Omron CX-Programmer project NewProject (CX-Programmer 9.87)

# PLC Teste: CP1L M

## Global symbols (name address type ; comment)
D315 CHANNEL  ; fim dm de contagem
Banco_de_Dados_29 Contador_de_Peças_PH29
Banco_de_Dados_30 Contador_de_Peças_PH30
Banco_de_Dados_31 Contador_de_Peças_PH31
Banco_de_Dados_F17 Contador_de_Peças_F17
Banco_de_Dados_F18 Contador_de_Peças_F18
Banco_de_Dados_F22 Contador_de_Peças_F22
Banco_de_Dados_R42 Contador_de_Peças_RC42
Banco_de_Dados_R43 Contador_de_Peças_RC43
Banco_de_dados_R41 Contador_de_Peças_RC41
Conta_Peças Contador_de_Peças_PH31
Visual_Formato_Trabalho_29 Formato_de_Trabalho_29
Visual_Formato_Trabalho_30 Formato_de_Trabalho_30
Visual_Formato_Trabalho_31 Formato_de_Trabalho_31

## Program Prensa (cyclic task 0)
Local symbols
F_31dias_vezes_2_ph30 D546 WORD
F_31dias_vezes_2_ph31 D530 WORD
F_Memoria_contagem_BCD_ph30 D552 WORD
F_Memoria_contagem_BCD_ph31 D536 WORD
F_Memória_de_Armazenagem_ph30 D550 WORD
F_Memória_de_Armazenagem_ph31 D534 WORD
F_Ponteiro_Dword_ph30 D548 WORD
F_Ponteiro_Dword_ph31 D532 WORD
KEEP 10.04 BOOL
MemAtuaReloSupervisorio H10.01 BOOL  ; Memória Atualiza Relogio pelo supervisório
Memoria_contagem_BCD_ph29 D528 WORD
Memoria_contagem_BCD_ph30 D518 WORD
Memoria_contagem_BCD_ph31 D508 WORD
Memoria_contagem_BIN_ph29 D526 WORD
Memoria_contagem_BIN_ph30 D516 WORD
Memoria_contagem_BIN_ph31 D506 WORD
Memória_de_Armazenagem_ph29 D524 WORD
Memória_de_Armazenagem_ph30 D514 WORD
Memória_de_Armazenagem_ph31 D504 WORD
PH29paradaT1 D0 CHANNEL  ; cnt prensa 31 parada T1
PH29paradaT2 D6 CHANNEL  ; cnt prensa 31 parada T2
PH29paradaT3 D12 CHANNEL  ; cnt prensa 31 parada T3
PH30paradaT1 D2 CHANNEL  ; cnt prensa 31 parada T1
PH30paradaT2 D8 CHANNEL  ; cnt prensa 31 parada T2
PH30paradaT3 D14 CHANNEL  ; cnt prensa 31 parada T3
PH31paradaT1 D4 CHANNEL  ; cnt prensa 31 parada T1
PH31paradaT2 D10 CHANNEL  ; cnt prensa 31 parada T2
PH31paradaT3 D18 CHANNEL  ; cnt prensa 31 parada T3
Ponteiro_Dword_ph29 D522 WORD
Ponteiro_Dword_ph30 D512 WORD
Ponteiro_Dword_ph31 D502 WORD
_31dias_vezes_2_ph29 D520 WORD
_31dias_vezes_2_ph30 D510 WORD
_31dias_vezes_2_ph31 D500 WORD
anoRelogio D36 CHANNEL  ; Ano Relógio
codFormPH29 D54 CHANNEL  ; Codigo do formato ph29
codFormPH30 D50 CHANNEL  ; Codigo do formato ph30
codFormPH31 D46 CHANNEL  ; Codigo do formato ph31
delayCicloPrensa29 T0001 BOOL  ; Retardo ciclo da prensa
delayCicloPrensa30 T0002 BOOL  ; Retardo ciclo da prensa
delayCicloPrensa31 T0003 BOOL  ; Retardo ciclo da prensa
diaCalendario D64 CHANNEL  ; dia calendario
diaMes D40 CHANNEL  ; dia do mes
diaRelogio D32 CHANNEL  ; Dia Relógio
filtroCntPc29 T0004 BOOL  ; filtro contagem peças
filtroCntPc30 T0005 BOOL  ; filtro contagem peças
filtroCntPc31 T0006 BOOL  ; filtro contagem peças
firstDMenvioFormat D56 CHANNEL  ; primeiro DM envio formato
firstDMenvioPcPH D42 CHANNEL  ; pirmeiro DM de envio peças ph
horaRelogio D30 CHANNEL  ; Horas Relogio
horas D58 CHANNEL  ; horas
iniciaCntTurno1 H10.02 BOOL  ; inicia contagem turno 1
iniciaCntTurno2 H10.03 BOOL  ; inicia contagem turno 2
iniciaCntTurno3 H10.04 BOOL  ; iniio contagem turno 3
linhaSelect D70 CHANNEL  ; linha selecionada
mesCalendario D66 CHANNEL  ; mes calendario
mesRelogio D34 CHANNEL  ; Mes Relogio
mesSelecionado D68 CHANNEL  ; mês selecionado
mesSelect D72 CHANNEL  ; mês selecionado
minutos D60 CHANNEL  ; minutos
minutosRelogio D28 CHANNEL  ; Minutos Relógio
numberCavidPH29 D52 CHANNEL  ; Número cavidades na prensa29
numberCavidPH30 D48 CHANNEL  ; Número cavidades na prensa30
numberCavidPH31 D44 CHANNEL  ; Número cavidades na prensa31
pecaPH29 D20 CHANNEL  ; conta peças ph29
pecaPH30 D22 CHANNEL  ; conta peças ph30
pecaPH31 D24 CHANNEL  ; conta peças ph31
ph29parada 10.00 BOOL  ; prensa 29 parada
ph30parada 10.01 BOOL  ; prensa 30 parada
ph31parada 10.03 BOOL  ; prensa 31 parada
ponteiroBDph29 D528 WORD  ; ponteiro banco de dados PH 29
ponteiroBDph30 D518 CHANNEL  ; ponteiro em BCD para armazenar a contagem
ponteiroBDph31 D508 WORD  ; ponteiro banco de dados PH31
prensa29 0.02 BOOL  ; Prensa 29
prensa30 0.01 BOOL  ; Prensa 30
prensa31 0.00 BOOL  ; Prensa 31
relogio4dig D38 CHANNEL  ; Ano Relógio 4 digitos
segundos D62 CHANNEL  ; segundos
segundosRelogio D26 CHANNEL  ; Segundos Relógio

### Section Reset

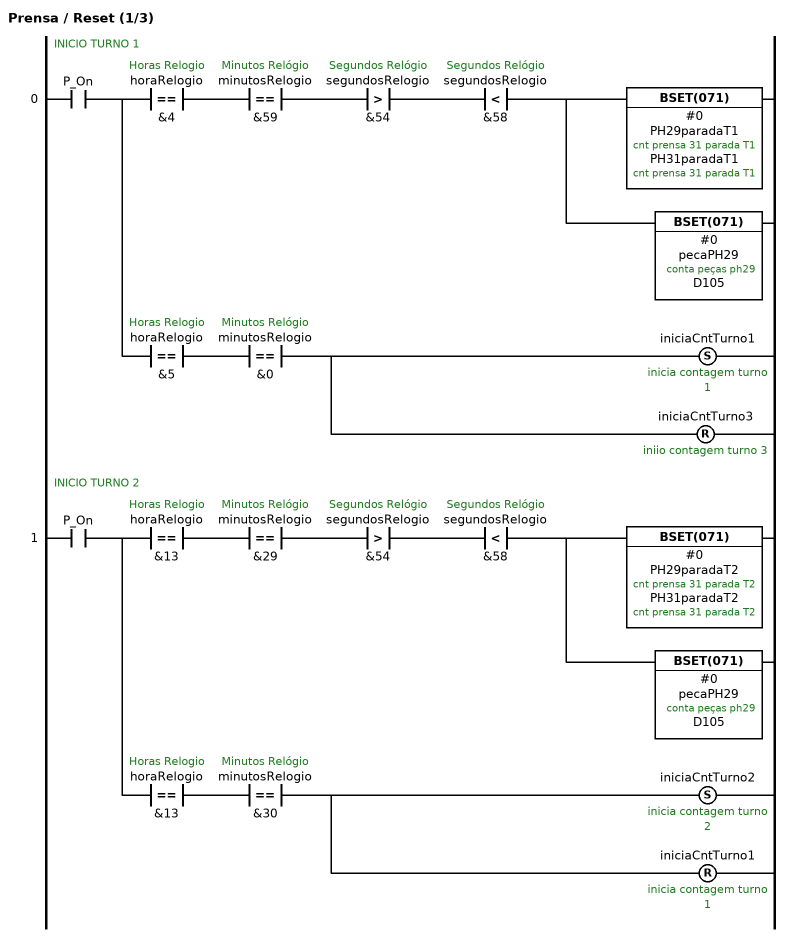
; rung 0: INICIO TURNO 1
LD P_On
OUT TR0
AND=(300) horaRelogio &4  ; Horas Relogio
AND=(300) minutosRelogio &59  ; Minutos Relógio
AND>(320) segundosRelogio &54  ; Segundos Relógio
AND<(310) segundosRelogio &58  ; Segundos Relógio
BSET(071) #0 PH29paradaT1 PH31paradaT1  ; cnt prensa 31 parada T1
BSET(071) #0 pecaPH29 D105  ; conta peças ph29
LD TR0
AND=(300) horaRelogio &5  ; Horas Relogio
AND=(300) minutosRelogio &0  ; Minutos Relógio
SET iniciaCntTurno1  ; inicia contagem turno 1
RSET iniciaCntTurno3  ; iniio contagem turno 3
; rung 1: INICIO TURNO 2
LD P_On
OUT TR0
AND=(300) horaRelogio &13  ; Horas Relogio
AND=(300) minutosRelogio &29  ; Minutos Relógio
AND>(320) segundosRelogio &54  ; Segundos Relógio
AND<(310) segundosRelogio &58  ; Segundos Relógio
BSET(071) #0 PH29paradaT2 PH31paradaT2  ; cnt prensa 31 parada T2
BSET(071) #0 pecaPH29 D105  ; conta peças ph29
LD TR0
AND=(300) horaRelogio &13  ; Horas Relogio
AND=(300) minutosRelogio &30  ; Minutos Relógio
SET iniciaCntTurno2  ; inicia contagem turno 2
RSET iniciaCntTurno1  ; inicia contagem turno 1

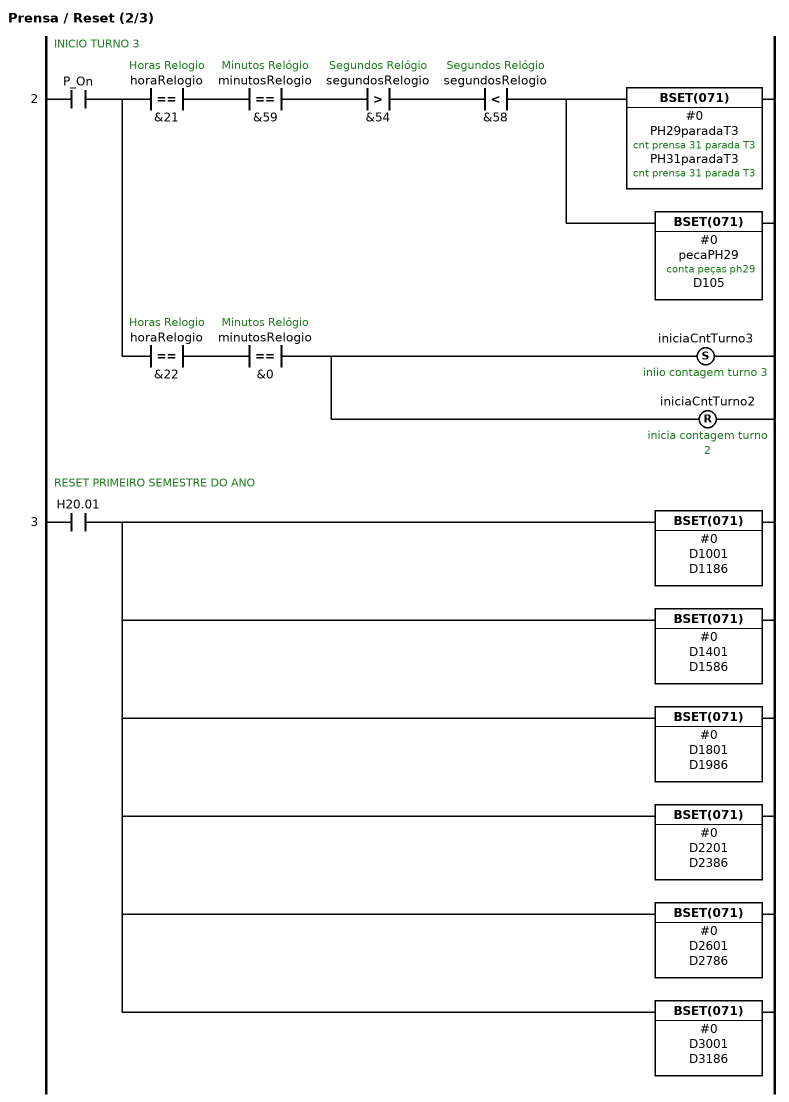
; rung 2: INICIO TURNO 3
LD P_On
OUT TR0
AND=(300) horaRelogio &21  ; Horas Relogio
AND=(300) minutosRelogio &59  ; Minutos Relógio
AND>(320) segundosRelogio &54  ; Segundos Relógio
AND<(310) segundosRelogio &58  ; Segundos Relógio
BSET(071) #0 PH29paradaT3 PH31paradaT3  ; cnt prensa 31 parada T3
BSET(071) #0 pecaPH29 D105  ; conta peças ph29
LD TR0
AND=(300) horaRelogio &22  ; Horas Relogio
AND=(300) minutosRelogio &0  ; Minutos Relógio
SET iniciaCntTurno3  ; iniio contagem turno 3
RSET iniciaCntTurno2  ; inicia contagem turno 2
; rung 3: RESET PRIMEIRO SEMESTRE DO ANO
LD H20.01
BSET(071) #0 D1001 D1186  // RESET PH31, 01/01 ATÉ 31/06
BSET(071) #0 D1401 D1586  // RESET PH30, 01/01 ATÉ 31/06
BSET(071) #0 D1801 D1986  // RESET PH29, 01/01 ATÉ 31/06
BSET(071) #0 D2201 D2386  // RESET FORMATO PH31, 01/01 ATÉ 31/06
BSET(071) #0 D2601 D2786  // RESET FORMATO PH30, 01/01 ATÉ 31/06
BSET(071) #0 D3001 D3186  // RESET FORMATO PH29, 01/01 ATÉ 31/06

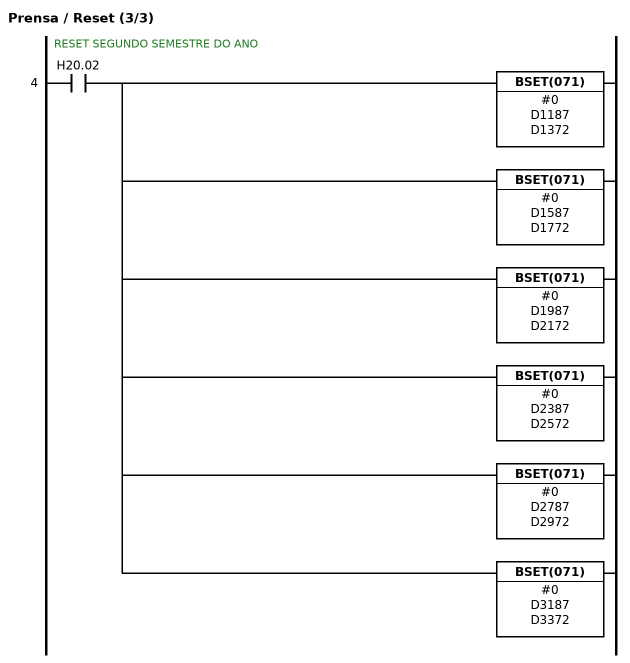
; rung 4: RESET SEGUNDO SEMESTRE DO ANO
LD H20.02
BSET(071) #0 D1187 D1372  // RESET PH31, 01/07 ATÉ 31/12
BSET(071) #0 D1587 D1772  // RESET PH30, 01/07 ATÉ 31/12
BSET(071) #0 D1987 D2172  // RESET PH29, 01/07 ATÉ 31/12
BSET(071) #0 D2387 D2572  // RESET FORMATO PH31, 01/07 ATÉ 31/12
BSET(071) #0 D2787 D2972  // RESET FORMATO PH30, 01/07 ATÉ 31/12
BSET(071) #0 D3187 D3372  // RESET FORMATO PH29, 01/07 ATÉ 31/12

### Section PH29

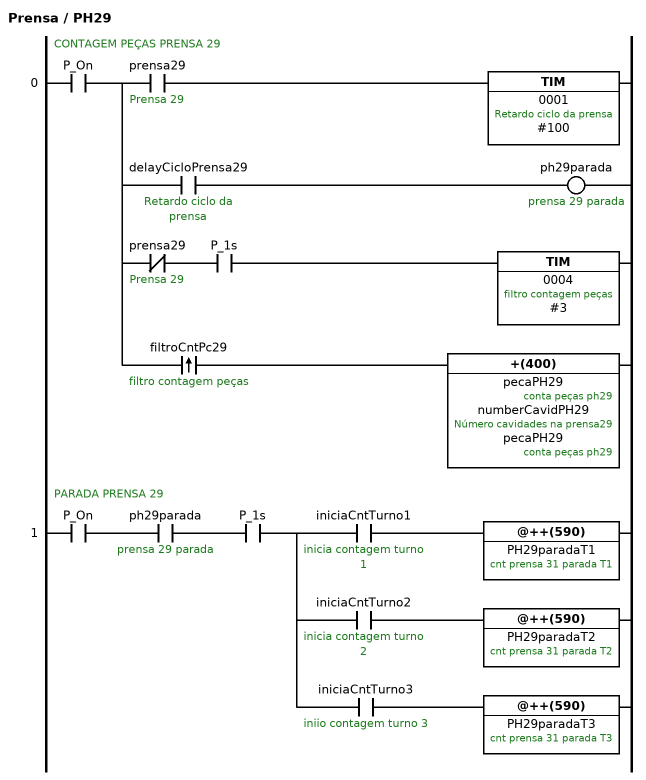
; rung 0: CONTAGEM PEÇAS PRENSA 29
LD P_On
OUT TR0
AND prensa29  ; Prensa 29
TIM 0001 #100  ; Retardo ciclo da prensa
LD TR0
AND delayCicloPrensa29  ; Retardo ciclo da prensa
OUT ph29parada  ; prensa 29 parada
LD TR0
ANDNOT prensa29  ; Prensa 29
AND P_1s
TIM 0004 #3  ; filtro contagem peças
LD TR0
@AND filtroCntPc29  ; filtro contagem peças
+(400) pecaPH29 numberCavidPH29 pecaPH29  ; conta peças ph29, Número cavidades na prensa29
; rung 1: PARADA PRENSA 29
LD P_On
AND ph29parada  ; prensa 29 parada
AND P_1s
OUT TR0
AND iniciaCntTurno1  ; inicia contagem turno 1
@++(590) PH29paradaT1  ; cnt prensa 31 parada T1  // CONTA PARADA TURNO 1
LD TR0
AND iniciaCntTurno2  ; inicia contagem turno 2
@++(590) PH29paradaT2  ; cnt prensa 31 parada T2  // CONTA PARADA TURNO 2
LD TR0
AND iniciaCntTurno3  ; iniio contagem turno 3
@++(590) PH29paradaT3  ; cnt prensa 31 parada T3  // CONTA PARADA TURNO 3

### Section PH30

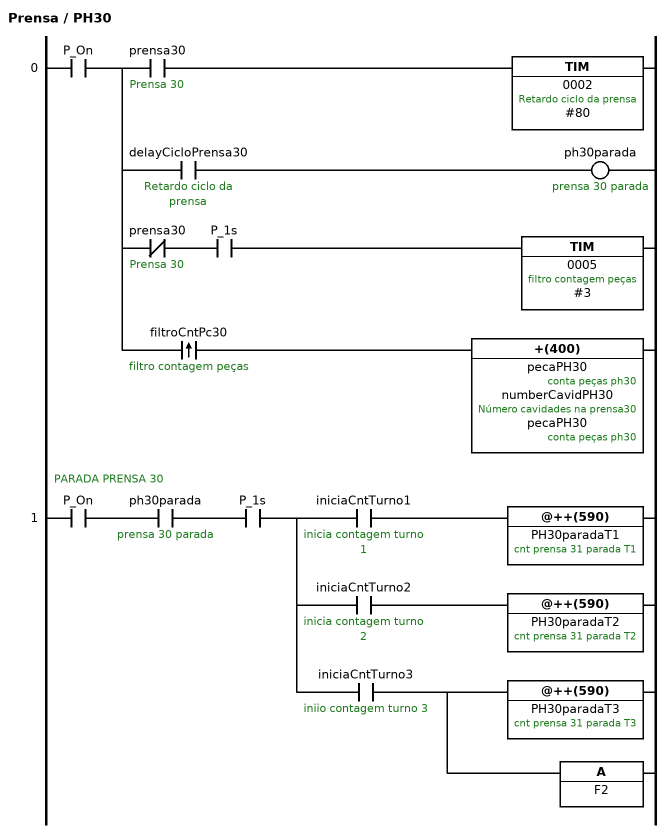
; rung 0
LD P_On
OUT TR0
AND prensa30  ; Prensa 30
TIM 0002 #80  ; Retardo ciclo da prensa
LD TR0
AND delayCicloPrensa30  ; Retardo ciclo da prensa
OUT ph30parada  ; prensa 30 parada
LD TR0
ANDNOT prensa30  ; Prensa 30
AND P_1s
TIM 0005 #3  ; filtro contagem peças
LD TR0
@AND filtroCntPc30  ; filtro contagem peças
+(400) pecaPH30 numberCavidPH30 pecaPH30  ; conta peças ph30, Número cavidades na prensa30
; rung 1: PARADA PRENSA 30
LD P_On  // D20 CONTA TURNO 2
AND ph30parada  ; prensa 30 parada
AND P_1s
OUT TR0
AND iniciaCntTurno1  ; inicia contagem turno 1
@++(590) PH30paradaT1  ; cnt prensa 31 parada T1
LD TR0
AND iniciaCntTurno2  ; inicia contagem turno 2
@++(590) PH30paradaT2  ; cnt prensa 31 parada T2
LD TR0
AND iniciaCntTurno3  ; iniio contagem turno 3
@++(590) PH30paradaT3  ; cnt prensa 31 parada T3  // D18 CONTA TURNO 1
A  F2
// D22 CONTA TURNO 3

### Section PH31

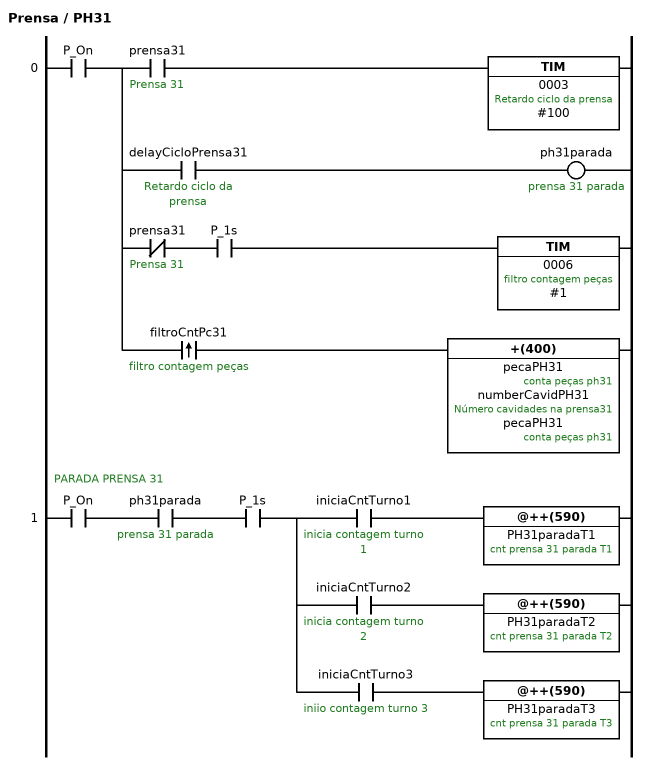
; rung 0
LD P_On
OUT TR0
AND prensa31  ; Prensa 31
TIM 0003 #100  ; Retardo ciclo da prensa
LD TR0
AND delayCicloPrensa31  ; Retardo ciclo da prensa
OUT ph31parada  ; prensa 31 parada
LD TR0
ANDNOT prensa31  ; Prensa 31
AND P_1s
TIM 0006 #1  ; filtro contagem peças
LD TR0
@AND filtroCntPc31  ; filtro contagem peças
+(400) pecaPH31 numberCavidPH31 pecaPH31  ; conta peças ph31, Número cavidades na prensa31
; rung 1: PARADA PRENSA 31
LD P_On
AND ph31parada  ; prensa 31 parada
AND P_1s
OUT TR0
AND iniciaCntTurno1  ; inicia contagem turno 1
@++(590) PH31paradaT1  ; cnt prensa 31 parada T1  // CONTA PARADA TURNO 1
LD TR0
AND iniciaCntTurno2  ; inicia contagem turno 2
@++(590) PH31paradaT2  ; cnt prensa 31 parada T2  // CONTA PARADA TURNO 2
LD TR0
AND iniciaCntTurno3  ; iniio contagem turno 3
@++(590) PH31paradaT3  ; cnt prensa 31 parada T3  // CONTA PARADA TUNOR 3

### Section Banco_de_Dados

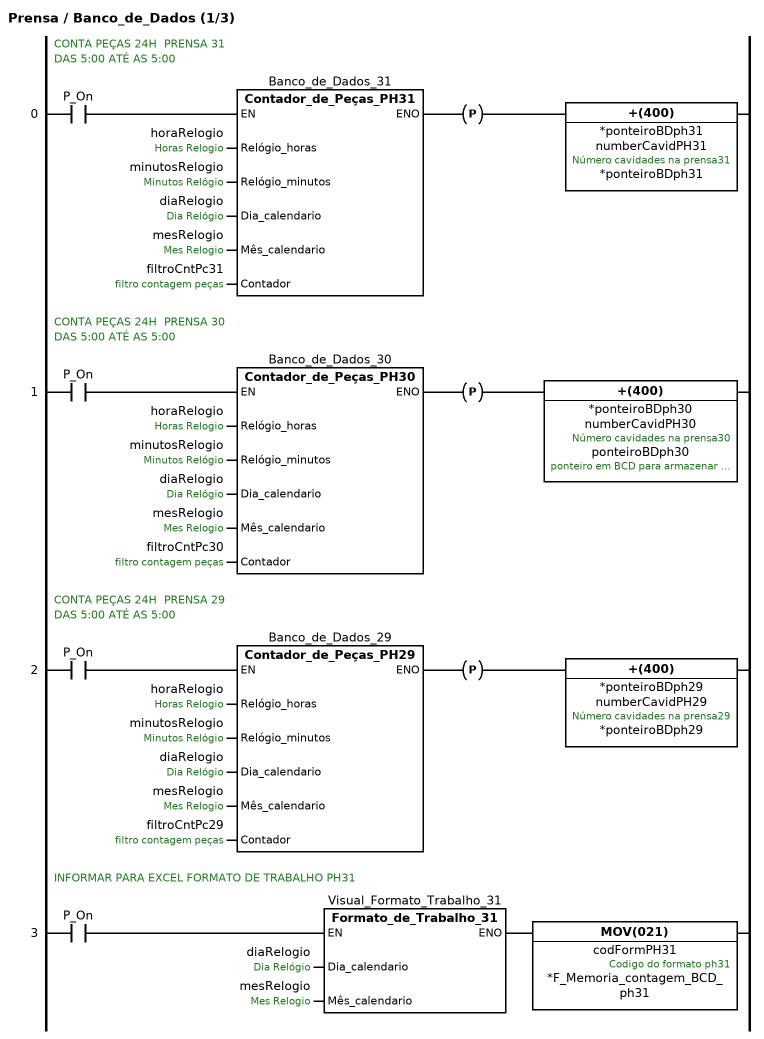
; rung 0: CONTA PEÇAS 24H  PRENSA 31 / DAS 5:00 ATÉ AS 5:00
LD P_On
CALL Banco_de_Dados_31 : Contador_de_Peças_PH31 (Relógio_horas := horaRelogio, Relógio_minutos := minutosRelogio, Dia_calendario := diaRelogio, Mês_calendario := mesRelogio, Contador := filtroCntPc31)  ; Horas Relogio, Minutos Relógio, Dia Relógio, Mes Relogio, filtro contagem peças
UP(521)
+(400) *ponteiroBDph31 numberCavidPH31 *ponteiroBDph31  ; Número cavidades na prensa31
; rung 1: CONTA PEÇAS 24H  PRENSA 30 / DAS 5:00 ATÉ AS 5:00
LD P_On
CALL Banco_de_Dados_30 : Contador_de_Peças_PH30 (Relógio_horas := horaRelogio, Relógio_minutos := minutosRelogio, Dia_calendario := diaRelogio, Mês_calendario := mesRelogio, Contador := filtroCntPc30)  ; Horas Relogio, Minutos Relógio, Dia Relógio, Mes Relogio, filtro contagem peças
UP(521)
+(400) *ponteiroBDph30 numberCavidPH30 ponteiroBDph30  ; Número cavidades na prensa30, ponteiro em BCD para armazenar a contagem
; rung 2: CONTA PEÇAS 24H  PRENSA 29 / DAS 5:00 ATÉ AS 5:00
LD P_On
CALL Banco_de_Dados_29 : Contador_de_Peças_PH29 (Relógio_horas := horaRelogio, Relógio_minutos := minutosRelogio, Dia_calendario := diaRelogio, Mês_calendario := mesRelogio, Contador := filtroCntPc29)  ; Horas Relogio, Minutos Relógio, Dia Relógio, Mes Relogio, filtro contagem peças
UP(521)
+(400) *ponteiroBDph29 numberCavidPH29 *ponteiroBDph29  ; Número cavidades na prensa29
; rung 3: INFORMAR PARA EXCEL FORMATO DE TRABALHO PH31
LD P_On
CALL Visual_Formato_Trabalho_31 : Formato_de_Trabalho_31 (Dia_calendario := diaRelogio, Mês_calendario := mesRelogio)  ; Dia Relógio, Mes Relogio
MOV(021) codFormPH31 *F_Memoria_contagem_BCD_ph31  ; Codigo do formato ph31

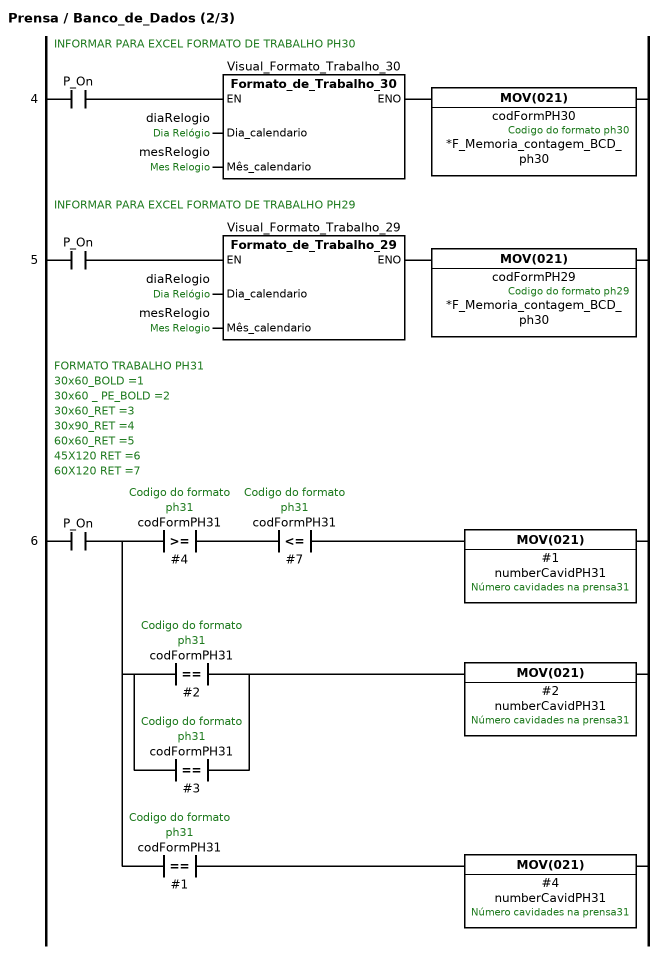
; rung 4: INFORMAR PARA EXCEL FORMATO DE TRABALHO PH30
LD P_On
CALL Visual_Formato_Trabalho_30 : Formato_de_Trabalho_30 (Dia_calendario := diaRelogio, Mês_calendario := mesRelogio)  ; Dia Relógio, Mes Relogio
MOV(021) codFormPH30 *F_Memoria_contagem_BCD_ph30  ; Codigo do formato ph30
; rung 5: INFORMAR PARA EXCEL FORMATO DE TRABALHO PH29
LD P_On
CALL Visual_Formato_Trabalho_29 : Formato_de_Trabalho_29 (Dia_calendario := diaRelogio, Mês_calendario := mesRelogio)  ; Dia Relógio, Mes Relogio
MOV(021) codFormPH29 *F_Memoria_contagem_BCD_ph30  ; Codigo do formato ph29
; rung 6: FORMATO TRABALHO PH31 / 30x60_BOLD =1 / 30x60_PE_BOLD =2 / 30x60_RET =3 / 30x90_RET =4 / 60x60_RET =5 / 45X120 RET =6 / 60X120 RET =7
LD P_On
OUT TR0
AND>=(325) codFormPH31 #4  ; Codigo do formato ph31
AND<=(315) codFormPH31 #7  ; Codigo do formato ph31
MOV(021) #1 numberCavidPH31  ; Número cavidades na prensa31
LD TR0
LD=(300) codFormPH31 #2  ; Codigo do formato ph31
OR=(300) codFormPH31 #3  ; Codigo do formato ph31
ANDLD
MOV(021) #2 numberCavidPH31  ; Número cavidades na prensa31
LD TR0
AND=(300) codFormPH31 #1  ; Codigo do formato ph31
MOV(021) #4 numberCavidPH31  ; Número cavidades na prensa31

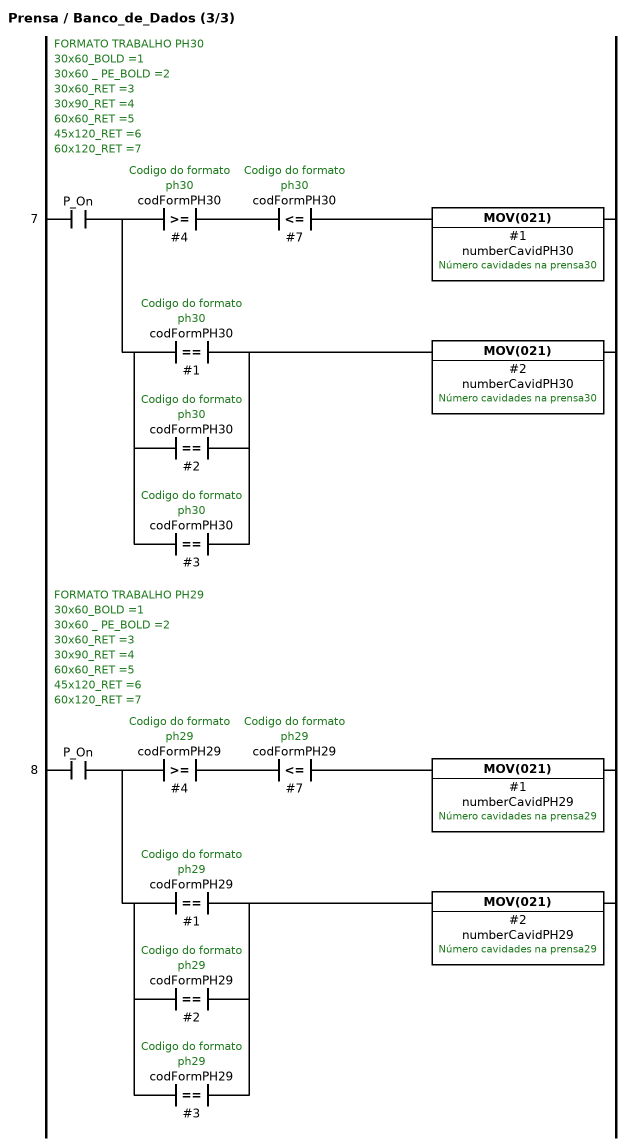
; rung 7: FORMATO TRABALHO PH30 / 30x60_BOLD =1 / 30x60_PE_BOLD =2 / 30x60_RET =3 / 30x90_RET =4 / 60x60_RET =5 / 45x120_RET =6 / 60x120_RET =7
LD P_On
OUT TR0
AND>=(325) codFormPH30 #4  ; Codigo do formato ph30
AND<=(315) codFormPH30 #7  ; Codigo do formato ph30
MOV(021) #1 numberCavidPH30  ; Número cavidades na prensa30
LD TR0
LD=(300) codFormPH30 #1  ; Codigo do formato ph30
OR=(300) codFormPH30 #2  ; Codigo do formato ph30
OR=(300) codFormPH30 #3  ; Codigo do formato ph30
ANDLD
MOV(021) #2 numberCavidPH30  ; Número cavidades na prensa30
; rung 8: FORMATO TRABALHO PH29 / 30x60_BOLD =1 / 30x60_PE_BOLD =2 / 30x60_RET =3 / 30x90_RET =4 / 60x60_RET =5 / 45x120_RET =6 / 60x120_RET =7
LD P_On
OUT TR0
AND>=(325) codFormPH29 #4  ; Codigo do formato ph29
AND<=(315) codFormPH29 #7  ; Codigo do formato ph29
MOV(021) #1 numberCavidPH29  ; Número cavidades na prensa29
LD TR0
LD=(300) codFormPH29 #1  ; Codigo do formato ph29
OR=(300) codFormPH29 #2  ; Codigo do formato ph29
OR=(300) codFormPH29 #3  ; Codigo do formato ph29
ANDLD
MOV(021) #2 numberCavidPH29  ; Número cavidades na prensa29

### Section Transferencia_excel

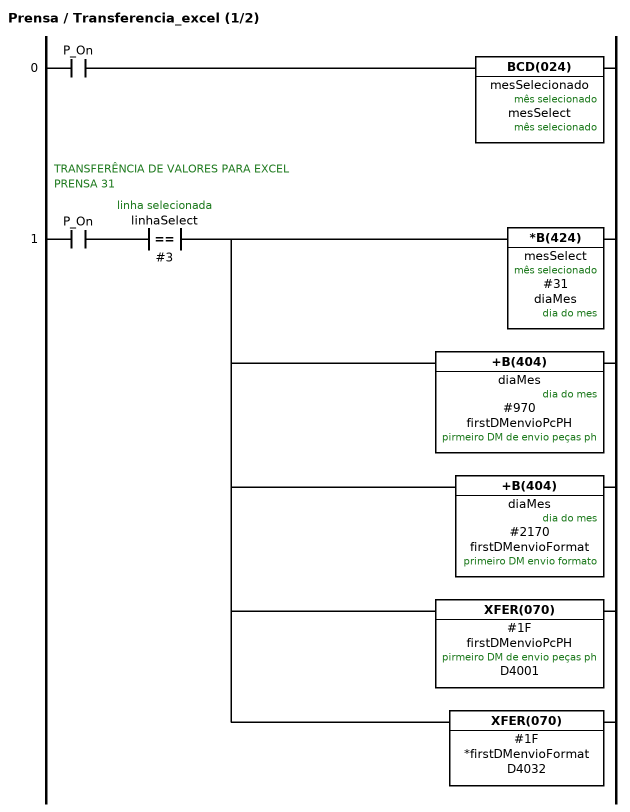
; rung 0
LD P_On
BCD(024) mesSelecionado mesSelect  ; mês selecionado
; rung 1: TRANSFERÊNCIA DE VALORES PARA EXCEL / PRENSA 31
LD P_On
AND=(300) linhaSelect #3  ; linha selecionada
*B(424) mesSelect #31 diaMes  ; mês selecionado, dia do mes  // SELECIONA O MES MULTIPLICA POR 31
+B(404) diaMes #970 firstDMenvioPcPH  ; dia do mes, pirmeiro DM de envio peças ph  // NUMERO DE DIAS DO ANO MULTIPLICA 970
+B(404) diaMes #2170 firstDMenvioFormat  ; dia do mes, primeiro DM envio formato
XFER(070) #1F firstDMenvioPcPH D4001  ; pirmeiro DM de envio peças ph  // TRANSFERE 31 DM APARTIR DO PRIMEIRO DM DE ENVIO
XFER(070) #1F *firstDMenvioFormat D4032

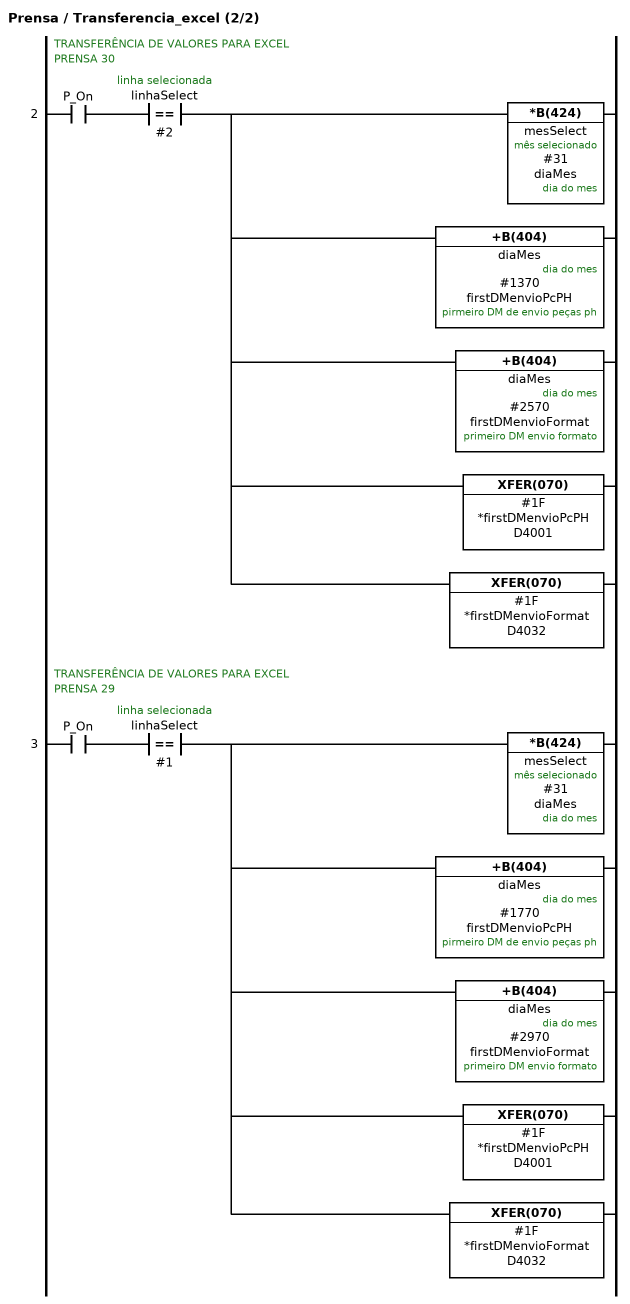
; rung 2: TRANSFERÊNCIA DE VALORES PARA EXCEL / PRENSA 30
LD P_On
AND=(300) linhaSelect #2  ; linha selecionada
*B(424) mesSelect #31 diaMes  ; mês selecionado, dia do mes
+B(404) diaMes #1370 firstDMenvioPcPH  ; dia do mes, pirmeiro DM de envio peças ph
+B(404) diaMes #2570 firstDMenvioFormat  ; dia do mes, primeiro DM envio formato
XFER(070) #1F *firstDMenvioPcPH D4001
XFER(070) #1F *firstDMenvioFormat D4032
; rung 3: TRANSFERÊNCIA DE VALORES PARA EXCEL / PRENSA 29
LD P_On
AND=(300) linhaSelect #1  ; linha selecionada
*B(424) mesSelect #31 diaMes  ; mês selecionado, dia do mes
+B(404) diaMes #1770 firstDMenvioPcPH  ; dia do mes, pirmeiro DM de envio peças ph
+B(404) diaMes #2970 firstDMenvioFormat  ; dia do mes, primeiro DM envio formato
XFER(070) #1F *firstDMenvioPcPH D4001
XFER(070) #1F *firstDMenvioFormat D4032

### Section Relogio

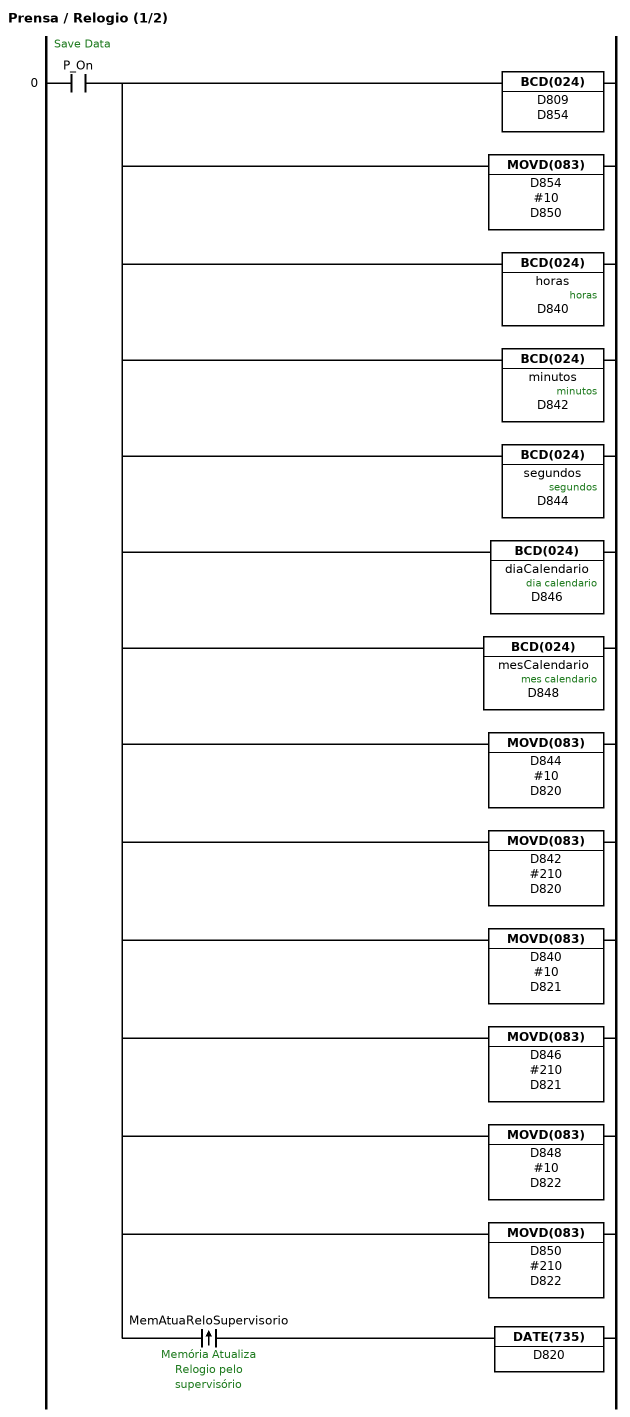
; rung 0: Save Data
LD P_On
BCD(024) D809 D854
MOVD(083) D854 #10 D850
BCD(024) horas D840  ; horas
BCD(024) minutos D842  ; minutos
BCD(024) segundos D844  ; segundos
BCD(024) diaCalendario D846  ; dia calendario
BCD(024) mesCalendario D848  ; mes calendario
MOVD(083) D844 #10 D820
MOVD(083) D842 #210 D820
MOVD(083) D840 #10 D821
MOVD(083) D846 #210 D821
MOVD(083) D848 #10 D822
MOVD(083) D850 #210 D822
@AND MemAtuaReloSupervisorio  ; Memória Atualiza Relogio pelo supervisório
DATE(735) D820

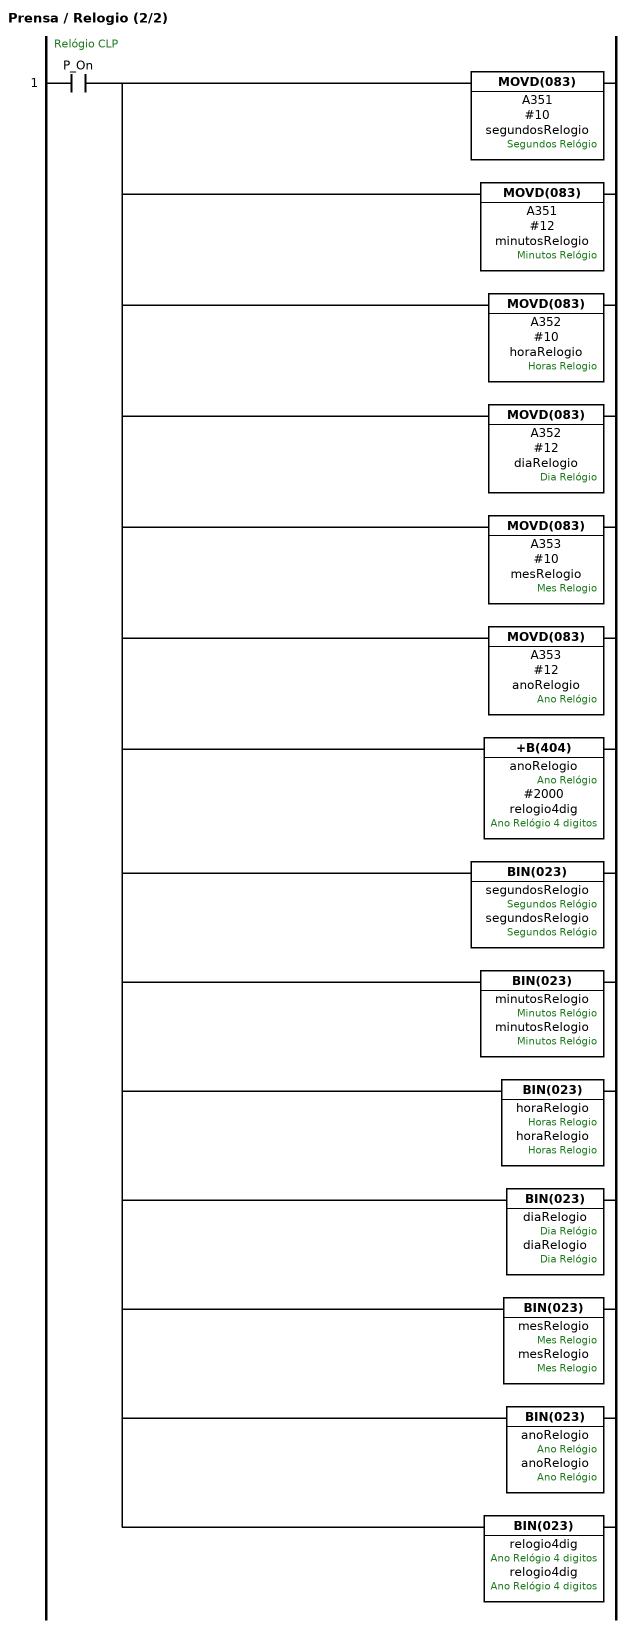
; rung 1: Relógio CLP
LD P_On
MOVD(083) A351 #10 segundosRelogio  ; Segundos Relógio
MOVD(083) A351 #12 minutosRelogio  ; Minutos Relógio
MOVD(083) A352 #10 horaRelogio  ; Horas Relogio
MOVD(083) A352 #12 diaRelogio  ; Dia Relógio
MOVD(083) A353 #10 mesRelogio  ; Mes Relogio
MOVD(083) A353 #12 anoRelogio  ; Ano Relógio
+B(404) anoRelogio #2000 relogio4dig  ; Ano Relógio, Ano Relógio 4 digitos
BIN(023) segundosRelogio segundosRelogio  ; Segundos Relógio
BIN(023) minutosRelogio minutosRelogio  ; Minutos Relógio
BIN(023) horaRelogio horaRelogio  ; Horas Relogio
BIN(023) diaRelogio diaRelogio  ; Dia Relógio
BIN(023) mesRelogio mesRelogio  ; Mes Relogio
BIN(023) anoRelogio anoRelogio  ; Ano Relógio
BIN(023) relogio4dig relogio4dig  ; Ano Relógio 4 digitos

### Section END
; rung 0
END(001)

## Program Carga (cyclic task 1)
Local symbols
AnoRelogio4dig_ D155 CHANNEL  ; Ano Relogio 4 Digitos
AnoRelógio4dit D156 CHANNEL  ; Ano Relógio 4 digitos
EnviRelogioSupervisorio H20.00 BOOL  ; Envia relogio superviório
HfornComForno18 H19.01 BOOL  ; forno com espaço
HfornoComEspacoF22 H19.02 BOOL  ; forno com espaço
HoraRelogio D163 CHANNEL  ; Horas Relogio
HrollerC42 H19.03 BOOL  ; roller carga 42
HrollerCarg43 H19.04 BOOL  ; roller carga 43
HrollerDesc41 H19.05 BOOL  ; roller descarga 41
HstatusRollerDesc41 H19.06 BOOL  ; status roller carga 41
HstatusRollerDesc42 H19.07 BOOL  ; status roller descarga 42
_d_segundos D150 CHANNEL  ; segundos
_r_horas D151 CHANNEL  ; horas
_t_minutos D152 CHANNEL  ; minutos
anoRelogio D153 CHANNEL  ; Ano Relógio
anoRelogio_ D154 CHANNEL  ; Ano Relógio
bancBaixoF18 40.06 BOOL  ; bancalino baixo carga forno 18
bancEntradaForno22 40.10 BOOL  ; bancalino entrada forno
cntContPc D157 CHANNEL  ; contador peças
cntPlanos43 C43 CHANNEL  ; contador de planos da 43
cntPlanosCargaRoller41 41.00 BOOL  ; contagem de planos da carga carro
cntPlanosCargaRoller42 41.02 BOOL  ; contador de gavetas carga roller mf42
cntPlanosDescRolle41 41.05 BOOL  ; contagem de planos da descarga carro
cntPlanosRollerCarga43 40.08 BOOL  ; cnt de planos de carga 43
cntPlanosRollerDescarga42 41.04 BOOL  ; contador descarga gaveta roller descarga mf42
cntPlanosRollerDescarga43 40.09 BOOL  ; cnt de planos de descarga 43
contPeçasCarga43 41.08 BOOL  ; contagem peças roller carga 43
corrEstoqIHMmenos41 H20.01 BOOL  ; correção estoque IHM (menos)
corrEstoqueIHM41 H19.15 BOOL  ; correção estoque IHM (mais)
corrEstoqueIHMmais41 H20.07 BOOL  ; correcão estoque(mais)
corrEstoqueIHMmais42 H20.03 BOOL  ; correção estoque IHM (mais)
corrEstoqueIHMmais43 H20.05 BOOL  ; correção estoque IHM (mais)
corrEstoqueIHMmenos41 H20.02 BOOL  ; correção estoque IHM (menos)
corrEstoqueIHMmenos42 H20.04 BOOL  ; correção estoque IHM (menos)
corrEstoqueIHMmenos43 H20.06 BOOL  ; correcão estoque(menos)
corrEstoqueMais42 H20.09 BOOL  ; correcão estoque(mais)
corrEstoqueMais43 H20.11 BOOL  ; correcão estoque(mais)
corrEstoqueMenos41 H20.08 BOOL  ; correcão estoque(menos)
corrEstoqueMenos42 H20.10 BOOL  ; correcão estoque(menos)
diaCalend D158 CHANNEL  ; dia calendario
diaMes D159 CHANNEL  ; dia do mes
diaRelogio D160 CHANNEL  ; Dia Relógio
estoqueVazio41 30.02 BOOL  ; estoque vazio
estoqueVazio42 30.04 BOOL  ; estoque zero mf42
estoqueVazio43 30.05 BOOL  ; comparador planos  vazios
filtroSen T0010 BOOL  ; filtro senso
firstDMenvioRoller D161 CHANNEL  ; primeiro DM envio roller
firstDMforno D162 CHANNEL  ; primeiro DM de contagem forno
fornoComEspacoF17 H19.00 BOOL  ; forno com espaço
ftcEspacoF17 40.03 BOOL  ; rele espaco forno 17 (saida 3.03)
ftcRolosForno17 40.02 BOOL  ; sensor sobre rolos entrada forno
iniciaCntT1 H19.08 BOOL  ; inicia contagem turno 1
iniciaCntT2 H19.09 BOOL  ; inicia contagem turno 2
iniciaCntT3 H19.10 BOOL  ; iniio contagem turno 3
ligaCnt10 50.00 BOOL  ; liga cnt10
ligaCnt11 50.02 BOOL  ; liga cnt11
ligaCnt12 50.04 BOOL  ; liga cnt12
linhaSelecionada D164 CHANNEL  ; linha selecionada
mesRelogio D166 CHANNEL  ; Mes Relogio
mesSelecionado D167 CHANNEL  ; mês selecionado
mesSelection D168 CHANNEL  ; mês selecionado
minRelogio D169 CHANNEL  ; Minutos Relógio
mêsCalend D165 CHANNEL  ; mês calendario
passoFormFila41 40.00 BOOL  ; passo a passo formador fila entrada roler 41
passoFormFila42 40.04 BOOL  ; passo a passo formador fila entrada roler 42
pcRollerDesc41 40.01 BOOL  ; sensor peças maquineta descarga 41
pecaFilaEntForno41 D170 CHANNEL  ; peças por fila entrada forno
peçaPorF17 D171 CHANNEL  ; peças por fila f17
peçaPorF18 D172 CHANNEL  ; peças por fila f18
peçaPorF22 D173 CHANNEL  ; peças por fila f22
ponteiroDB22 D174 CHANNEL
receitaDestF22 D3800 CHANNEL  ; receita de destino F22
receitaDestRolle43 D3001 CHANNEL  ; receita de destino RC43
releF18 40.07 BOOL  ; rele forno 18 (saida 3.03)
releF22 40.11 BOOL  ; rele forno 22
reseRetornoPc1 20.00 BOOL  ; reset retorno peças
reseRetornoPc2 20.01 BOOL  ; reset retorno peças
reseRetornoPc3 20.02 BOOL  ; reset retorno peças
resetCnt10 50.01 BOOL  ; reset cnt10
resetCnt11 50.03 BOOL  ; reset cnt11
resetCnt12 50.05 BOOL  ; reset cnt12
resetInicioT1 C0010 BOOL  ; reset inicio turno 1
resetInicioT2 C0011 BOOL  ; reset inicio turno 2
resetInicioT3 C0012 BOOL  ; reset inicio turno 3
segRelogio D205 CHANNEL  ; Segundos Relógio
statusRollDesc43 H19.11 BOOL  ; status roller descarga 43
statusRollerCarg41 41.03 BOOL  ; status roller C41
statusRollerCarga43 41.09 BOOL  ; status roller C43
statusRollerDesc41 41.01 BOOL  ; status roller C41
statusRollerDesc42 40.05 BOOL  ; status roller desc. 42
statusRollerDesc43 H19.12 BOOL  ; status roller descarga 43
turno1_2_3 D175 CHANNEL  ; turno 1,2,3

### Section Principal

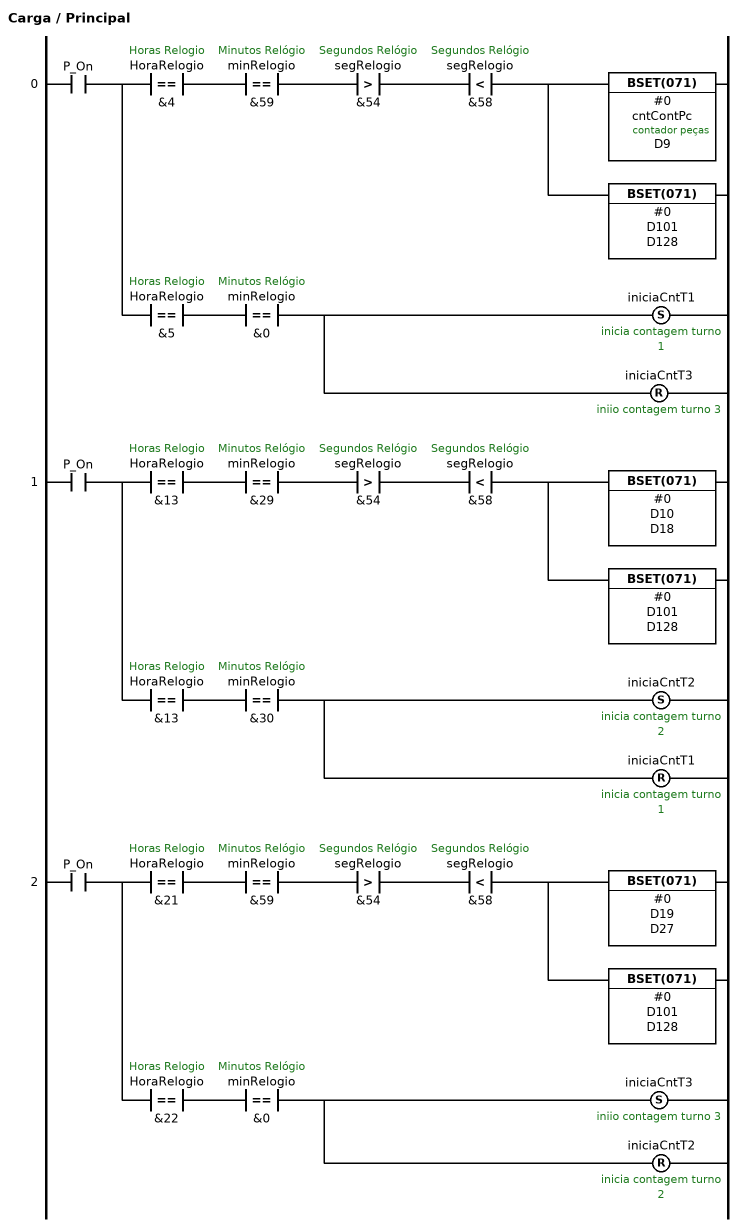
; rung 0
LD P_On
OUT TR0
AND=(300) HoraRelogio &4  ; Horas Relogio
AND=(300) minRelogio &59  ; Minutos Relógio
AND>(320) segRelogio &54  ; Segundos Relógio
AND<(310) segRelogio &58  ; Segundos Relógio
BSET(071) #0 cntContPc D9  ; contador peças
BSET(071) #0 D101 D128
LD TR0
AND=(300) HoraRelogio &5  ; Horas Relogio
AND=(300) minRelogio &0  ; Minutos Relógio
SET iniciaCntT1  ; inicia contagem turno 1
RSET iniciaCntT3  ; iniio contagem turno 3
; rung 1
LD P_On
OUT TR0
AND=(300) HoraRelogio &13  ; Horas Relogio
AND=(300) minRelogio &29  ; Minutos Relógio
AND>(320) segRelogio &54  ; Segundos Relógio
AND<(310) segRelogio &58  ; Segundos Relógio
BSET(071) #0 D10 D18
BSET(071) #0 D101 D128
LD TR0
AND=(300) HoraRelogio &13  ; Horas Relogio
AND=(300) minRelogio &30  ; Minutos Relógio
SET iniciaCntT2  ; inicia contagem turno 2
RSET iniciaCntT1  ; inicia contagem turno 1
; rung 2
LD P_On
OUT TR0
AND=(300) HoraRelogio &21  ; Horas Relogio
AND=(300) minRelogio &59  ; Minutos Relógio
AND>(320) segRelogio &54  ; Segundos Relógio
AND<(310) segRelogio &58  ; Segundos Relógio
BSET(071) #0 D19 D27
BSET(071) #0 D101 D128
LD TR0
AND=(300) HoraRelogio &22  ; Horas Relogio
AND=(300) minRelogio &0  ; Minutos Relógio
SET iniciaCntT3  ; iniio contagem turno 3
RSET iniciaCntT2  ; inicia contagem turno 2

### Section MF41

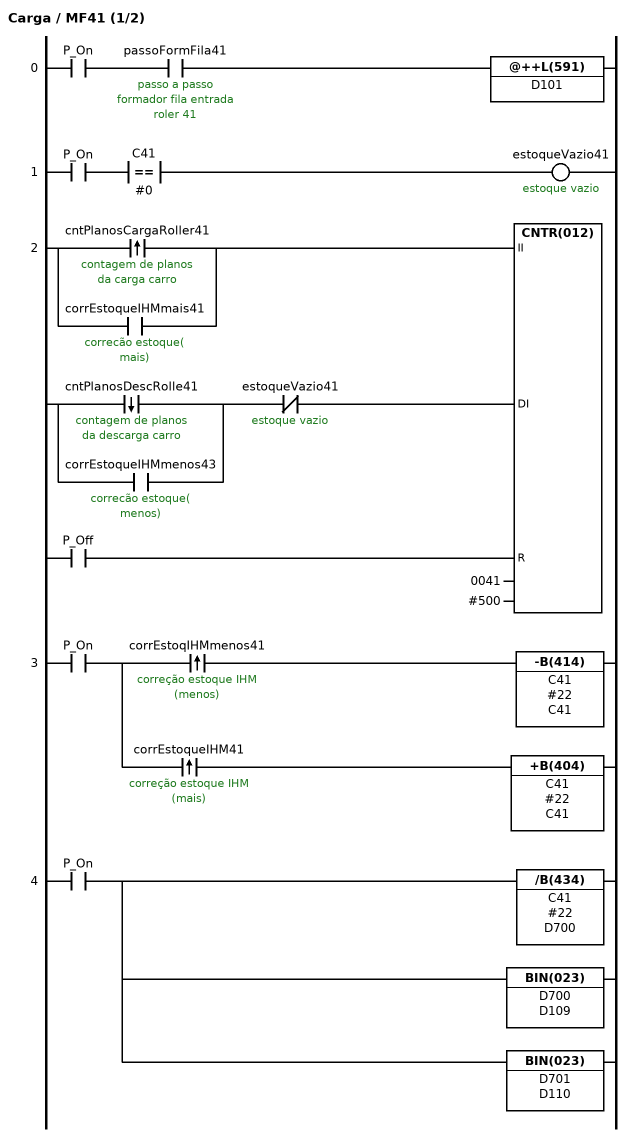
; rung 0
LD P_On
AND passoFormFila41  ; passo a passo formador fila entrada roler 41
@++L(591) D101
; rung 1
LD P_On
AND=(300) C41 #0
OUT estoqueVazio41  ; estoque vazio
; rung 2
@LD cntPlanosCargaRoller41  ; contagem de planos da carga carro
OR corrEstoqueIHMmais41  ; correcão estoque(mais)
%LD cntPlanosDescRolle41  ; contagem de planos da descarga carro
OR corrEstoqueIHMmenos43  ; correcão estoque(menos)
ANDNOT estoqueVazio41  ; estoque vazio
LD P_Off
CNTR(012) 0041 #500
; rung 3
LD P_On
OUT TR0
@AND corrEstoqIHMmenos41  ; correção estoque IHM (menos)
-B(414) C41 #22 C41
LD TR0
@AND corrEstoqueIHM41  ; correção estoque IHM (mais)
+B(404) C41 #22 C41
; rung 4
LD P_On
/B(434) C41 #22 D700
BIN(023) D700 D109
BIN(023) D701 D110

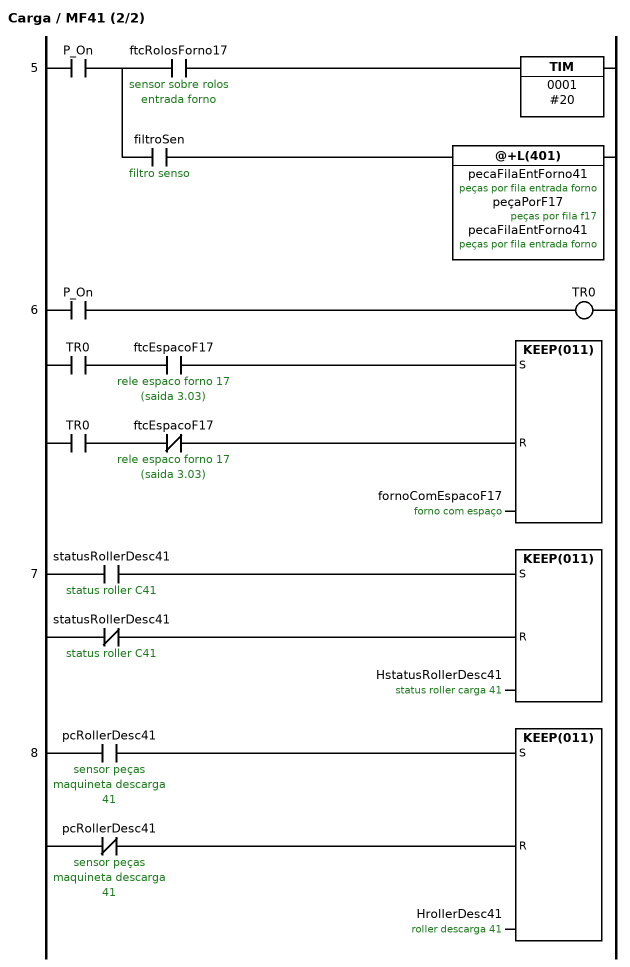
; rung 5
LD P_On
OUT TR0
AND ftcRolosForno17  ; sensor sobre rolos entrada forno
TIM 0001 #20
LD TR0
AND filtroSen  ; filtro senso
@+L(401) pecaFilaEntForno41 peçaPorF17 pecaFilaEntForno41  ; peças por fila entrada forno, peças por fila f17
; rung 6
LD P_On
OUT TR0
AND ftcEspacoF17  ; rele espaco forno 17 (saida 3.03)
LD TR0
ANDNOT ftcEspacoF17  ; rele espaco forno 17 (saida 3.03)
KEEP(011) fornoComEspacoF17  ; forno com espaço
; rung 7
LD statusRollerDesc41  ; status roller C41
LDNOT statusRollerDesc41  ; status roller C41
KEEP(011) HstatusRollerDesc41  ; status roller carga 41
; rung 8
LD pcRollerDesc41  ; sensor peças maquineta descarga 41
LDNOT pcRollerDesc41  ; sensor peças maquineta descarga 41
KEEP(011) HrollerDesc41  ; roller descarga 41

### Section MF42

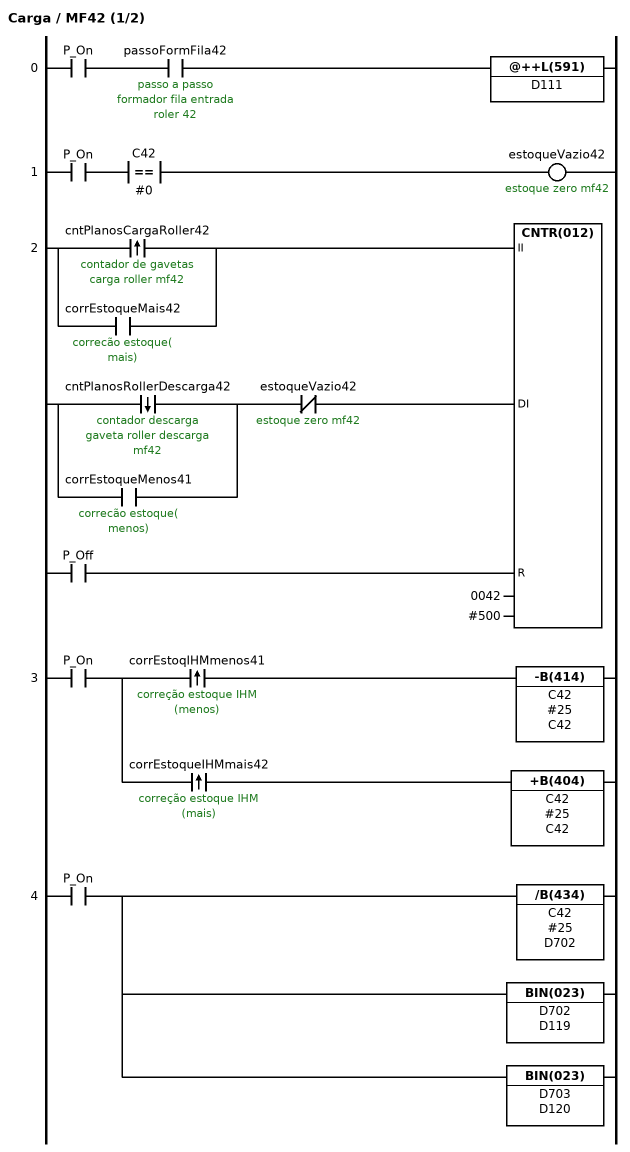
; rung 0
LD P_On
AND passoFormFila42  ; passo a passo formador fila entrada roler 42
@++L(591) D111
; rung 1
LD P_On
AND=(300) C42 #0
OUT estoqueVazio42  ; estoque zero mf42
; rung 2
@LD cntPlanosCargaRoller42  ; contador de gavetas carga roller mf42
OR corrEstoqueMais42  ; correcão estoque(mais)
%LD cntPlanosRollerDescarga42  ; contador descarga gaveta roller descarga mf42
OR corrEstoqueMenos41  ; correcão estoque(menos)
ANDNOT estoqueVazio42  ; estoque zero mf42
LD P_Off
CNTR(012) 0042 #500
; rung 3
LD P_On
OUT TR0
@AND corrEstoqIHMmenos41  ; correção estoque IHM (menos)
-B(414) C42 #25 C42
LD TR0
@AND corrEstoqueIHMmais42  ; correção estoque IHM (mais)
+B(404) C42 #25 C42
; rung 4
LD P_On
/B(434) C42 #25 D702
BIN(023) D702 D119
BIN(023) D703 D120

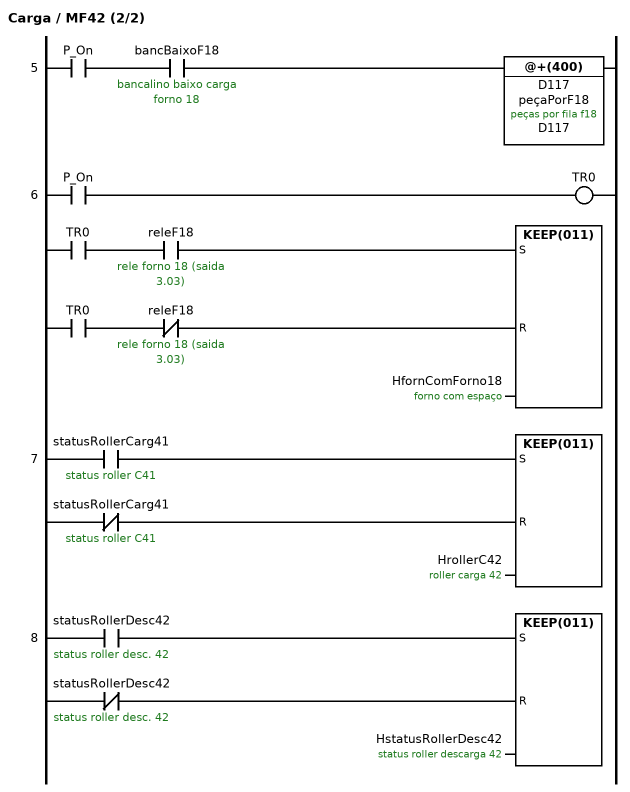
; rung 5
LD P_On
AND bancBaixoF18  ; bancalino baixo carga forno 18
@+(400) D117 peçaPorF18 D117  ; peças por fila f18
; rung 6
LD P_On
OUT TR0
AND releF18  ; rele forno 18 (saida 3.03)
LD TR0
ANDNOT releF18  ; rele forno 18 (saida 3.03)
KEEP(011) HfornComForno18  ; forno com espaço
; rung 7
LD statusRollerCarg41  ; status roller C41
LDNOT statusRollerCarg41  ; status roller C41
KEEP(011) HrollerC42  ; roller carga 42
; rung 8
LD statusRollerDesc42  ; status roller desc. 42
LDNOT statusRollerDesc42  ; status roller desc. 42
KEEP(011) HstatusRollerDesc42  ; status roller descarga 42

### Section MF43

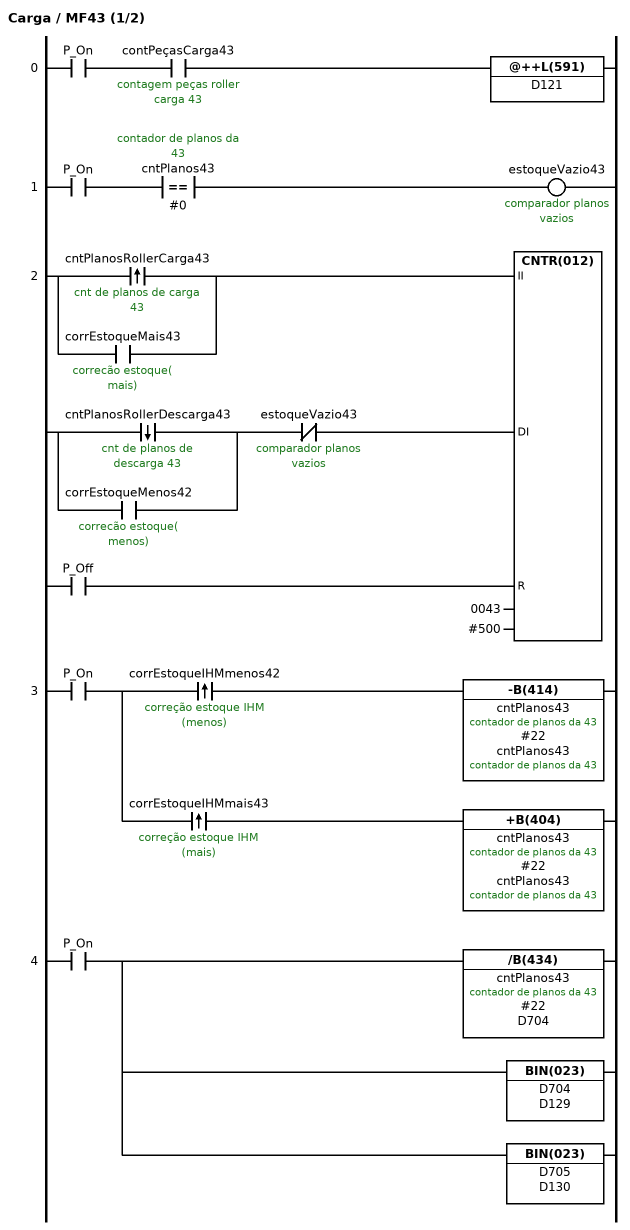
; rung 0
LD P_On
AND contPeçasCarga43  ; contagem peças roller carga 43
@++L(591) D121
; rung 1
LD P_On
AND=(300) cntPlanos43 #0  ; contador de planos da 43
OUT estoqueVazio43  ; comparador planos  vazios
; rung 2
@LD cntPlanosRollerCarga43  ; cnt de planos de carga 43
OR corrEstoqueMais43  ; correcão estoque(mais)
%LD cntPlanosRollerDescarga43  ; cnt de planos de descarga 43
OR corrEstoqueMenos42  ; correcão estoque(menos)
ANDNOT estoqueVazio43  ; comparador planos  vazios
LD P_Off
CNTR(012) 0043 #500
; rung 3
LD P_On
OUT TR0
@AND corrEstoqueIHMmenos42  ; correção estoque IHM (menos)
-B(414) cntPlanos43 #22 cntPlanos43  ; contador de planos da 43
LD TR0
@AND corrEstoqueIHMmais43  ; correção estoque IHM (mais)
+B(404) cntPlanos43 #22 cntPlanos43  ; contador de planos da 43
; rung 4
LD P_On
/B(434) cntPlanos43 #22 D704  ; contador de planos da 43
BIN(023) D704 D129
BIN(023) D705 D130

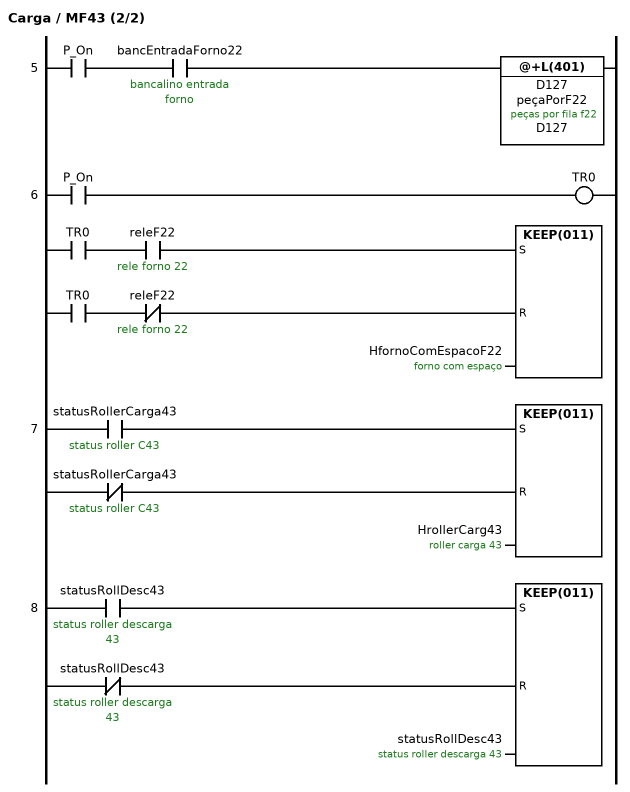
; rung 5
LD P_On
AND bancEntradaForno22  ; bancalino entrada forno
@+L(401) D127 peçaPorF22 D127  ; peças por fila f22
; rung 6
LD P_On
OUT TR0
AND releF22  ; rele forno 22
LD TR0
ANDNOT releF22  ; rele forno 22
KEEP(011) HfornoComEspacoF22  ; forno com espaço
; rung 7
LD statusRollerCarga43  ; status roller C43
LDNOT statusRollerCarga43  ; status roller C43
KEEP(011) HrollerCarg43  ; roller carga 43
; rung 8
LD statusRollDesc43  ; status roller descarga 43
LDNOT statusRollDesc43  ; status roller descarga 43
KEEP(011) statusRollDesc43  ; status roller descarga 43

### Section MF41_ESPAÇO

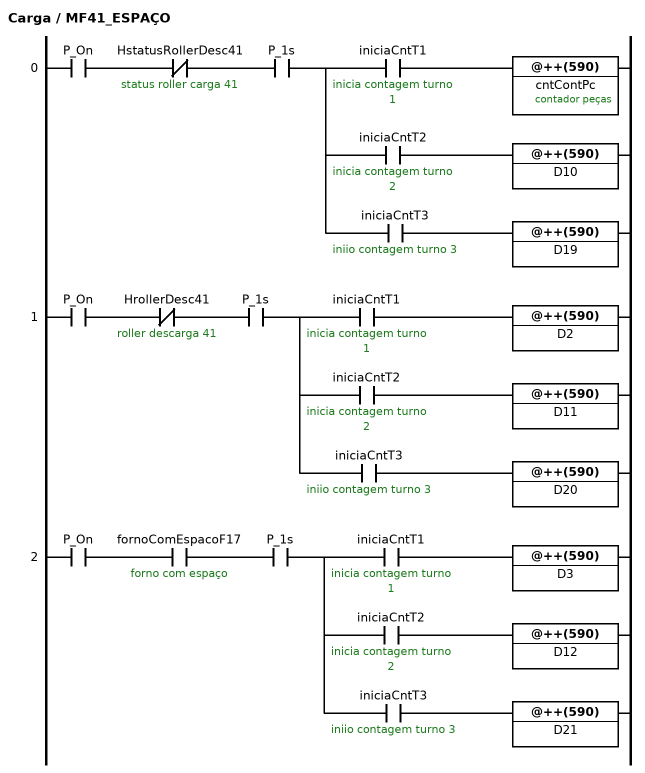
; rung 0
LD P_On
ANDNOT HstatusRollerDesc41  ; status roller carga 41
AND P_1s
OUT TR0
AND iniciaCntT1  ; inicia contagem turno 1
@++(590) cntContPc  ; contador peças
LD TR0
AND iniciaCntT2  ; inicia contagem turno 2
@++(590) D10
LD TR0
AND iniciaCntT3  ; iniio contagem turno 3
@++(590) D19
; rung 1
LD P_On
ANDNOT HrollerDesc41  ; roller descarga 41
AND P_1s
OUT TR0
AND iniciaCntT1  ; inicia contagem turno 1
@++(590) D2
LD TR0
AND iniciaCntT2  ; inicia contagem turno 2
@++(590) D11
LD TR0
AND iniciaCntT3  ; iniio contagem turno 3
@++(590) D20
; rung 2
LD P_On
AND fornoComEspacoF17  ; forno com espaço
AND P_1s
OUT TR0
AND iniciaCntT1  ; inicia contagem turno 1
@++(590) D3
LD TR0
AND iniciaCntT2  ; inicia contagem turno 2
@++(590) D12
LD TR0
AND iniciaCntT3  ; iniio contagem turno 3
@++(590) D21

### Section MF42_ESPAÇO

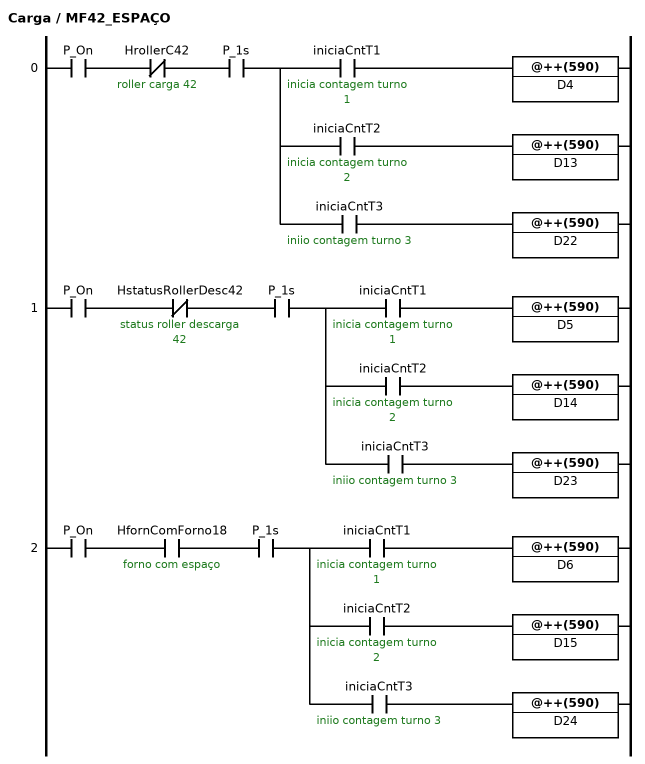
; rung 0
LD P_On
ANDNOT HrollerC42  ; roller carga 42
AND P_1s
OUT TR0
AND iniciaCntT1  ; inicia contagem turno 1
@++(590) D4
LD TR0
AND iniciaCntT2  ; inicia contagem turno 2
@++(590) D13
LD TR0
AND iniciaCntT3  ; iniio contagem turno 3
@++(590) D22
; rung 1
LD P_On
ANDNOT HstatusRollerDesc42  ; status roller descarga 42
AND P_1s
OUT TR0
AND iniciaCntT1  ; inicia contagem turno 1
@++(590) D5
LD TR0
AND iniciaCntT2  ; inicia contagem turno 2
@++(590) D14
LD TR0
AND iniciaCntT3  ; iniio contagem turno 3
@++(590) D23
; rung 2
LD P_On
AND HfornComForno18  ; forno com espaço
AND P_1s
OUT TR0
AND iniciaCntT1  ; inicia contagem turno 1
@++(590) D6
LD TR0
AND iniciaCntT2  ; inicia contagem turno 2
@++(590) D15
LD TR0
AND iniciaCntT3  ; iniio contagem turno 3
@++(590) D24

### Section MF43_ESPAÇO

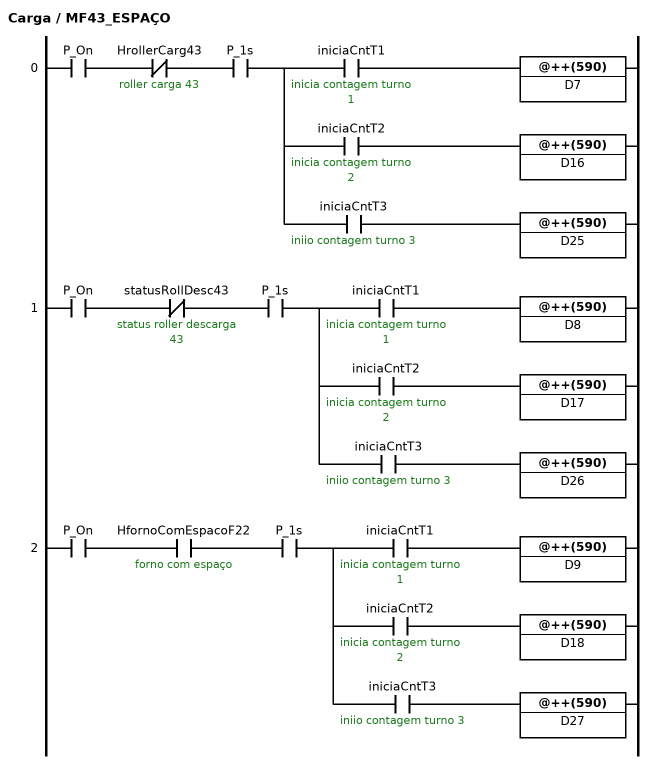
; rung 0
LD P_On
ANDNOT HrollerCarg43  ; roller carga 43
AND P_1s
OUT TR0
AND iniciaCntT1  ; inicia contagem turno 1
@++(590) D7
LD TR0
AND iniciaCntT2  ; inicia contagem turno 2
@++(590) D16
LD TR0
AND iniciaCntT3  ; iniio contagem turno 3
@++(590) D25
; rung 1
LD P_On
ANDNOT statusRollDesc43  ; status roller descarga 43
AND P_1s
OUT TR0
AND iniciaCntT1  ; inicia contagem turno 1
@++(590) D8
LD TR0
AND iniciaCntT2  ; inicia contagem turno 2
@++(590) D17
LD TR0
AND iniciaCntT3  ; iniio contagem turno 3
@++(590) D26
; rung 2
LD P_On
AND HfornoComEspacoF22  ; forno com espaço
AND P_1s
OUT TR0
AND iniciaCntT1  ; inicia contagem turno 1
@++(590) D9
LD TR0
AND iniciaCntT2  ; inicia contagem turno 2
@++(590) D18
LD TR0
AND iniciaCntT3  ; iniio contagem turno 3
@++(590) D27

### Section Banco_de_Dados

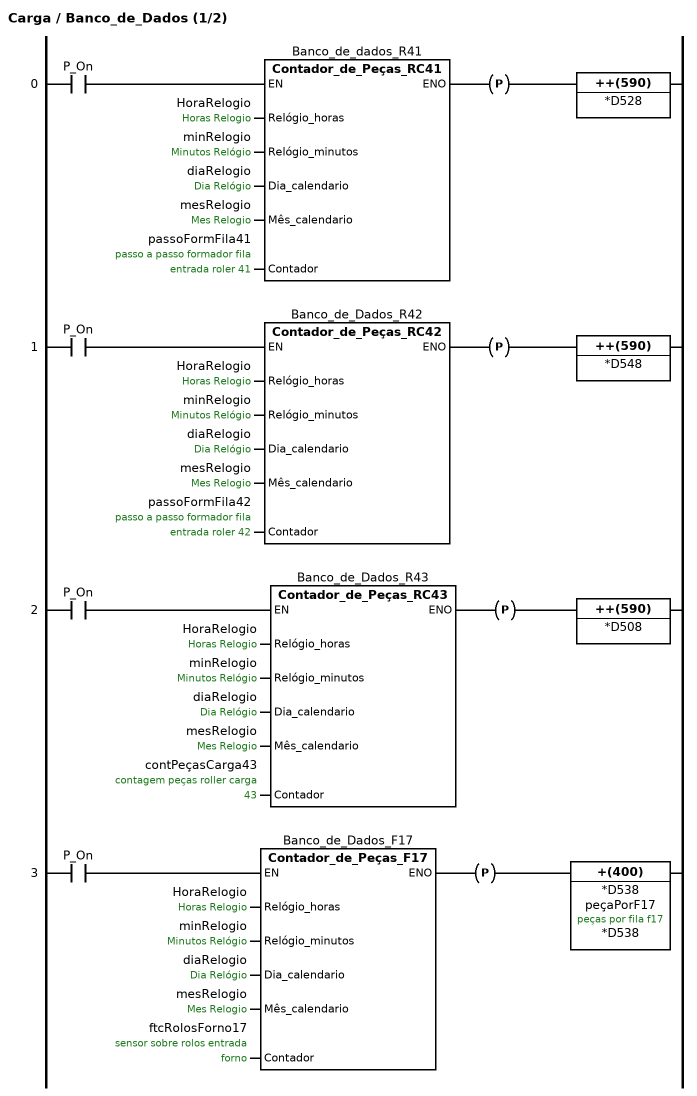
; rung 0
LD P_On
CALL Banco_de_dados_R41 : Contador_de_Peças_RC41 (Relógio_horas := HoraRelogio, Relógio_minutos := minRelogio, Dia_calendario := diaRelogio, Mês_calendario := mesRelogio, Contador := passoFormFila41)  ; Horas Relogio, Minutos Relógio, Dia Relógio, Mes Relogio, passo a passo formador fila entrada roler 41
UP(521)
++(590) *D528
; rung 1
LD P_On
CALL Banco_de_Dados_R42 : Contador_de_Peças_RC42 (Relógio_horas := HoraRelogio, Relógio_minutos := minRelogio, Dia_calendario := diaRelogio, Mês_calendario := mesRelogio, Contador := passoFormFila42)  ; Horas Relogio, Minutos Relógio, Dia Relógio, Mes Relogio, passo a passo formador fila entrada roler 42
UP(521)
++(590) *D548
; rung 2
LD P_On
CALL Banco_de_Dados_R43 : Contador_de_Peças_RC43 (Relógio_horas := HoraRelogio, Relógio_minutos := minRelogio, Dia_calendario := diaRelogio, Mês_calendario := mesRelogio, Contador := contPeçasCarga43)  ; Horas Relogio, Minutos Relógio, Dia Relógio, Mes Relogio, contagem peças roller carga 43
UP(521)
++(590) *D508
; rung 3
LD P_On
CALL Banco_de_Dados_F17 : Contador_de_Peças_F17 (Relógio_horas := HoraRelogio, Relógio_minutos := minRelogio, Dia_calendario := diaRelogio, Mês_calendario := mesRelogio, Contador := ftcRolosForno17)  ; Horas Relogio, Minutos Relógio, Dia Relógio, Mes Relogio, sensor sobre rolos entrada forno
UP(521)
+(400) *D538 peçaPorF17 *D538  ; peças por fila f17

